Staubli VAL3: create.pgx

public program create(num x_nEncNum (dimensions=1), string x_sTask (dimensions=1))
begin
  call init(x_nEncNum,x_sTask)
  taskCreate sTASK,100,encoder()
end
